{attribute 'qualified_only'}
VAR_GLOBAL
	arrServoCtrl			: ARRAY[0..gc.usiMaxNrOfAxes] OF typ_ServoIF;
END_VAR

(* stored: Version 1.1.0.1, ProductVersion 3.1.4022.17
   GVL gFB: Id {7a6ade20-3bbf-4ea4-bf9f-b6920edff0e2} *)
